FUNCTION_BLOCK FB_DS301_DS402_Object_Testing
VAR_INPUT
	NodeID			: BYTE; (* This Port No. addresses the CANopen Node (see System Manager) *)
	Start			: BOOL;
END_VAR
VAR_OUTPUT
	Finished		: BOOL;
END_VAR
VAR_IN_OUT
	CAN_Objects		: ARRAY [*] OF ST_CAN_Object_Test;
END_VAR
VAR
	State			: BYTE := 0;
	Index			: DINT := 0;
	
	NMT_WRITE		: FB_NMT_WRITE;
	
	SDO_READ		: FB_SDO_READ;
	ReadData		: ARRAY [0..255] OF BYTE;
	
	SDO_WRITE		: FB_SDO_WRITE;
	WriteData		: ARRAY [0..255] OF BYTE;		
			
	RPDO_Nr				: BYTE := 3;	
	RPDO_Current_Number	: BYTE := 0;
	RPDO_Current_Mapped	: DWORD := 0;	
	
	TPDO_Nr				: BYTE := 3;
	TPDO_Current_Number	: BYTE := 0;
	TPDO_Current_Mapped	: DWORD := 0;
END_VAR

IF Start AND State = 255 THEN 
	State := 0;
END_IF

SDO_READ(StartReading:=FALSE);
SDO_WRITE(StartWriting:=FALSE);
NMT_WRITE(StartWriting:=FALSE);


CASE State OF	
	// ********** Initial steps **********	
	0: // NMT Set to Preoperational
		NMT_WRITE(
			AdsNetID	:= '5.156.6.243.3.1',
			PortNr		:= 16#1000 + NodeID,
			ADSSTATE	:= ADSSTATE_RUN, 
			DEVSTATE	:= 0,
			StartWriting:=TRUE			
		);	
		
		IF NMT_WRITE.WriteDataFinished THEN
			Index := 0;	
			State := State + 1;	
		END_IF
		

	1:	// RPDO disable
		WriteData[3] := 16#80;
		WriteData[2] := 0;			
		WriteData[1] := RPDO_Nr + 1;
		WriteData[0] := NodeID;	
			
		SDO_WRITE(
			ADSNetID		:= '5.156.6.243.3.1',
			PortNr 		 	:= 16#1000 + NodeID,
			CO_Index 	 	:= 16#1400 + RPDO_Nr,
			CO_SubIndex  	:= 1,
			DataLength 	 	:= 4,
			StartWriting 	:= TRUE,
			WriteData 	 	:= WriteData );
		
		IF SDO_WRITE.WriteDataFinished THEN
			State := State + 1;
		END_IF	
		
		
	2:	// RPDO Current Number of mapped objects
		SDO_READ(
			ADSNetID		:= '5.156.6.243.3.1',				
			PortNr 		 	:= 16#1000 + NodeID,
			CO_Index 		:= 16#1600 + RPDO_Nr,
			CO_SubIndex 	:= 0,
			DataLength 		:= 1,
			StartReading	:= TRUE	);
		
		IF SDO_READ.ReadDataAvailable THEN
			RPDO_Current_Number := SDO_READ.ReadData[0];
			State := State + 1;
		END_IF
		
	
	3:	// RPDO Current mapped object
		SDO_READ(
			ADSNetID		:= '5.156.6.243.3.1',				
			PortNr 		 	:= 16#1000 + NodeID,
			CO_Index 		:= 16#1600 + RPDO_Nr,
			CO_SubIndex 	:= 1,
			DataLength 		:= 4,
			StartReading	:= TRUE	);
		
		IF SDO_READ.ReadDataAvailable THEN
			RPDO_Current_Mapped := SHL(BYTE_TO_DWORD(SDO_READ.ReadData[3]),24) + SHL(BYTE_TO_DWORD(SDO_READ.ReadData[2]),16) + SHL(BYTE_TO_DWORD(SDO_READ.ReadData[1]),8) + BYTE_TO_DWORD(SDO_READ.ReadData[0]);								
			State := State + 1;
		END_IF		
			
		
	4:	// TPDO disable
		WriteData[3] := 16#80;
		WriteData[2] := 0;			
		WriteData[1] := TPDO_Nr;
		WriteData[0] := NodeID + 16#80;	
			
		SDO_WRITE(
			ADSNetID		:= '5.156.6.243.3.1',
			PortNr 		 	:= 16#1000 + NodeID,
			CO_Index 	 	:= 16#1800 + TPDO_Nr,
			CO_SubIndex  	:= 1,
			DataLength 	 	:= 4,
			StartWriting 	:= TRUE,
			WriteData 	 	:= WriteData );
		
		IF SDO_WRITE.WriteDataFinished THEN
			State := State + 1;
		END_IF	
		

	5:	// TPDO Current Number of mapped objects
		SDO_READ(
			ADSNetID		:= '5.156.6.243.3.1',				
			PortNr 		 	:= 16#1000 + NodeID,
			CO_Index 		:= 16#1A00 + TPDO_Nr,
			CO_SubIndex 	:= 0,
			DataLength 		:= 1,
			StartReading	:= TRUE	);
		
		IF SDO_READ.ReadDataAvailable THEN
			TPDO_Current_Number := SDO_READ.ReadData[0];			
			State := State + 1;
		END_IF
		

	6:	// TPDO Current mapped object
		SDO_READ(
			ADSNetID		:= '5.156.6.243.3.1',				
			PortNr 		 	:= 16#1000 + NodeID,
			CO_Index 		:= 16#1A00 + TPDO_Nr,
			CO_SubIndex 	:= 1,
			DataLength 		:= 4,
			StartReading	:= TRUE	);
		
		IF SDO_READ.ReadDataAvailable THEN
			TPDO_Current_Mapped := SHL(BYTE_TO_DWORD(SDO_READ.ReadData[3]),24) + SHL(BYTE_TO_DWORD(SDO_READ.ReadData[2]),16) + SHL(BYTE_TO_DWORD(SDO_READ.ReadData[1]),8) + BYTE_TO_DWORD(SDO_READ.ReadData[0]);							
			State := 16;
		END_IF		
		
		
		
	// ********** Test steps **********
	16:	// Init
		CAN_Objects[Index].SDO_Read_Done := FALSE;
		CAN_Objects[Index].SDO_Read_Value := 0;				
		CAN_Objects[Index].SDO_Read_Error := 0;	
		CAN_Objects[Index].SDO_Write_Done := FALSE;			
		CAN_Objects[Index].SDO_Write_Error := 0;	
		CAN_Objects[Index].RPDO_Done := FALSE;			
		CAN_Objects[Index].RPDO_Error := 0;	
		CAN_Objects[Index].TPDO_Done := FALSE;			
		CAN_Objects[Index].TPDO_Error := 0;	

		// Transform value for Write Test
		WriteData[0] := DWORD_TO_BYTE(CAN_Objects[Index].SDO_Write_Value);
		WriteData[1] := DWORD_TO_BYTE(SHR(CAN_Objects[Index].SDO_Write_Value,8));
		WriteData[2] := DWORD_TO_BYTE(SHR(CAN_Objects[Index].SDO_Write_Value,16));
		WriteData[3] := DWORD_TO_BYTE(SHR(CAN_Objects[Index].SDO_Write_Value,24));
		
		State := State + 1;
			
		
	17:	// Read Test
		IF CAN_Objects[Index].CAN_Object.Readable THEN
			SDO_READ(
				ADSNetID		:= '5.156.6.243.3.1',				
				PortNr 		 	:= 16#1000 + NodeID,
				CO_Index 		:= CAN_Objects[Index].CAN_Object.Index,
				CO_SubIndex 	:= CAN_Objects[Index].CAN_Object.Subindex,
				DataLength 		:= CAN_Objects[Index].CAN_Object.Length,
				StartReading	:= TRUE	);
			
			IF SDO_READ.ReadDataAvailable THEN
				CAN_Objects[Index].SDO_Read_Done := TRUE;
				CAN_Objects[Index].SDO_Read_Value := SHL(BYTE_TO_DWORD(SDO_READ.ReadData[3]),24) + SHL(BYTE_TO_DWORD(SDO_READ.ReadData[2]),16) + SHL(BYTE_TO_DWORD(SDO_READ.ReadData[1]),8) + BYTE_TO_DWORD(SDO_READ.ReadData[0]);				
				CAN_Objects[Index].SDO_Read_Error := SDO_READ.Error;
				IF CAN_Objects[Index].WriteTest_with_CurrentValue THEN	
					WriteData := SDO_READ.ReadData; 
				END_IF			
		
				State := State + 1;
			END_IF
		ELSE
			// Not done -> Result
			CAN_Objects[Index].SDO_Read_Done := FALSE;
			CAN_Objects[Index].SDO_Read_Value := 0;				
			CAN_Objects[Index].SDO_Read_Error := 0;
						
			State := State + 1;	
		END_IF
	
		
	18:	// Write Test
		IF CAN_Objects[Index].CAN_Object.Writeable THEN
			SDO_WRITE(
				ADSNetID	:= '5.156.6.243.3.1',
				PortNr 		 := 16#1000 + NodeID,
				CO_Index 	 := CAN_Objects[Index].CAN_Object.Index,
				CO_SubIndex  := CAN_Objects[Index].CAN_Object.Subindex,
				DataLength 	 := CAN_Objects[Index].CAN_Object.Length,
				StartWriting := TRUE,
				WriteData 	 := WriteData );
			
			IF SDO_WRITE.WriteDataFinished THEN
				CAN_Objects[Index].SDO_Write_Done := TRUE;
				CAN_Objects[Index].SDO_Write_Value := SHL(BYTE_TO_DWORD(SDO_Write.WriteData[3]),24) + SHL(BYTE_TO_DWORD(SDO_Write.WriteData[2]),16) + SHL(BYTE_TO_DWORD(SDO_Write.WriteData[1]),8) + BYTE_TO_DWORD(SDO_Write.WriteData[0]);				
				CAN_Objects[Index].SDO_Write_Error := SDO_WRITE.Error;
				
				State := State + 1;
			END_IF
		ELSE
			CAN_Objects[Index].SDO_Write_Done := FALSE;
			CAN_Objects[Index].SDO_Write_Value := 0;				
			CAN_Objects[Index].SDO_Write_Error := 0;	
			
			State := State + 1;	
		END_IF			

		
	19: // RPDO test
		IF CAN_Objects[Index].CAN_Object.RPDO_Mappable THEN
			WriteData[0] := CAN_Objects[Index].CAN_Object.Length * 8;
			WriteData[1] := CAN_Objects[Index].CAN_Object.SubIndex;
			WriteData[2] := DWORD_TO_BYTE(CAN_Objects[Index].CAN_Object.Index);
			WriteData[3] := DWORD_TO_BYTE(SHR(CAN_Objects[Index].CAN_Object.Index,8));
		
			SDO_WRITE(
				ADSNetID	:= '5.156.6.243.3.1',
				PortNr 		 := 16#1000 + NodeID,
				CO_Index 	 := 16#1600 + RPDO_Nr,
				CO_SubIndex  := 1,
				DataLength 	 := 4,
				StartWriting := TRUE,
				WriteData 	 := WriteData );			
			
			IF SDO_WRITE.WriteDataFinished THEN
				CAN_Objects[Index].RPDO_Done := TRUE;
				CAN_Objects[Index].RPDO_Error := SDO_WRITE.Error;
				
				State := State + 1;
			END_IF
		ELSE
			CAN_Objects[Index].RPDO_Done := FALSE;	
			CAN_Objects[Index].RPDO_Error := 0;	
			
			State := State + 1;	
		END_IF			

				
	20: // TPDO test
		IF CAN_Objects[Index].CAN_Object.TPDO_Mappable THEN
			WriteData[0] := CAN_Objects[Index].CAN_Object.Length * 8;
			WriteData[1] := CAN_Objects[Index].CAN_Object.SubIndex;
			WriteData[2] := DWORD_TO_BYTE(CAN_Objects[Index].CAN_Object.Index);
			WriteData[3] := DWORD_TO_BYTE(SHR(CAN_Objects[Index].CAN_Object.Index,8));
		
			SDO_WRITE(
				ADSNetID	:= '5.156.6.243.3.1',
				PortNr 		 := 16#1000 + NodeID,
				CO_Index 	 := 16#1A00 + TPDO_Nr,
				CO_SubIndex  := 1,
				DataLength 	 := 4,
				StartWriting := TRUE,
				WriteData 	 := WriteData );			
			
		IF SDO_WRITE.WriteDataFinished THEN
				CAN_Objects[Index].TPDO_Done := TRUE;
				CAN_Objects[Index].TPDO_Error := SDO_WRITE.Error;
				
				State := State + 1;
			END_IF
		ELSE
			CAN_Objects[Index].TPDO_Done := FALSE;	
			CAN_Objects[Index].TPDO_Error := 0;	
			
			State := State + 1;	
		END_IF
		
		
	21: // Next object
		CAN_Objects[Index].Error := (CAN_Objects[Index].SDO_Read_Error > 0) OR (CAN_Objects[Index].SDO_Write_Error > 0) OR (CAN_Objects[Index].RPDO_Error > 0) OR (CAN_Objects[Index].TPDO_Error > 0);
			
		IF Index < UPPER_BOUND(CAN_Objects,1) THEN
			Index := Index + 1;
			State := 16;
		ELSE
			State := 50;
		END_IF
	
		
	// ********** Ending steps **********		
	50:	// RPDO Reset mapped object
		WriteData[0] := DWORD_TO_BYTE(RPDO_Current_Mapped);
		WriteData[1] := DWORD_TO_BYTE(SHR(RPDO_Current_Mapped,8));
		WriteData[2] := DWORD_TO_BYTE(SHR(RPDO_Current_Mapped,16));
		WriteData[3] := DWORD_TO_BYTE(SHR(RPDO_Current_Mapped,24));
		
		SDO_WRITE(
			ADSNetID		:= '5.156.6.243.3.1',			
			PortNr 		 	:= 16#1000 + NodeID,
			CO_Index 		:= 16#1600 + TPDO_Nr,
			CO_SubIndex 	:= 1,
			DataLength 		:= 4,
			StartWriting	:= TRUE,
			WriteData 	 	:= WriteData );
		
		IF SDO_WRITE.WriteDataFinished THEN
			State := State + 1;
		END_IF		
			
		
	51:	// RPDO Reset Number of mapped objects
		WriteData[0] := RPDO_Current_Number;
			
		SDO_WRITE(
			ADSNetID		:= '5.156.6.243.3.1',
			PortNr 		 	:= 16#1000 + NodeID,
			CO_Index 		:= 16#1600 + RPDO_Nr,
			CO_SubIndex 	:= 0,
			DataLength 		:= 1,
			StartWriting 	:= TRUE,
			WriteData 	 	:= WriteData );
		
		IF SDO_WRITE.WriteDataFinished THEN
			State := State + 1;
		END_IF			

		
	52:	// RPDO reactivate
		WriteData[3] := 0;
		WriteData[2] := 0;			
		WriteData[1] := RPDO_Nr + 1;
		WriteData[0] := NodeID;	
			
		SDO_WRITE(
			ADSNetID	:= '5.156.6.243.3.1',
			PortNr 		 := 16#1000 + NodeID,
			CO_Index 	 := 16#1400 + RPDO_Nr,
			CO_SubIndex  := 1,
			DataLength 	 := 4,
			StartWriting := TRUE,
			WriteData 	 := WriteData );
		
		IF SDO_WRITE.WriteDataFinished THEN
			State := State + 1;
		END_IF	
		
		
	53:	// TPDO Reset mapped object
		WriteData[0] := DWORD_TO_BYTE(TPDO_Current_Mapped);
		WriteData[1] := DWORD_TO_BYTE(SHR(TPDO_Current_Mapped,8));
		WriteData[2] := DWORD_TO_BYTE(SHR(TPDO_Current_Mapped,16));
		WriteData[3] := DWORD_TO_BYTE(SHR(TPDO_Current_Mapped,24));
		
		SDO_WRITE(
			ADSNetID		:= '5.156.6.243.3.1',			
			PortNr 		 	:= 16#1000 + NodeID,
			CO_Index 		:= 16#1A00 + TPDO_Nr,
			CO_SubIndex 	:= 1,
			DataLength 		:= 4,
			StartWriting	:= TRUE,
			WriteData 	 	:= WriteData );
		
		IF SDO_WRITE.WriteDataFinished THEN
			State := State + 1;
		END_IF			
			
		
	54:	// TPDO Reset Number of mapped objects
		WriteData[0] := TPDO_Current_Number;
			
		SDO_WRITE(
			ADSNetID		:= '5.156.6.243.3.1',
			PortNr 		 	:= 16#1000 + NodeID,
			CO_Index 		:= 16#1A00 + RPDO_Nr,
			CO_SubIndex 	:= 0,
			DataLength 		:= 1,
			StartWriting 	:= TRUE,
			WriteData 	 	:= WriteData );
		
		IF SDO_WRITE.WriteDataFinished THEN
			State := State + 1;
		END_IF			

		
	55:	// TPDO reactivate
		WriteData[3] := 0;
		WriteData[2] := 0;			
		WriteData[1] := TPDO_Nr;
		WriteData[0] := NodeID + 16#80;	
			
		SDO_WRITE(
			ADSNetID	:= '5.156.6.243.3.1',
			PortNr 		 := 16#1000 + NodeID,
			CO_Index 	 := 16#1400 + RPDO_Nr,
			CO_SubIndex  := 1,
			DataLength 	 := 4,
			StartWriting := TRUE,
			WriteData 	 := WriteData );
		
		IF SDO_WRITE.WriteDataFinished THEN
			State := State + 1;
		END_IF	
						
	
	56: // NMT Set to operational
		NMT_WRITE(
			ADSNetID	:= '5.156.6.243.3.1',
			PORTNr		:= 16#1000 + NodeID,
			ADSSTATE	:= ADSSTATE_RUN,
			DEVSTATE	:= 1,
			StartWriting:=TRUE );	
		
		IF NMT_WRITE.WriteDataFinished THEN
			State := 255;	
		END_IF

		
	// ********** End **********
	ELSE	// Tests finished	
		Finished := TRUE;
		State := 255;
			
END_CASE

END_FUNCTION_BLOCK

(* stored: Version 1.1.0.1, ProductVersion 3.1.4024.11
   POU FB_DS301_DS402_Object_Testing: Id {8bcecccf-0172-4904-a369-b9a49f46e69c}, SpecialFunc None *)
